Staubli VAL3: MoveLine.pgx

program MoveLine(num x_nX, num x_nY, num x_nZ, num x_nRx, num x_nRy, num x_nRz)
begin
  pPointRx1.trsf.x = x_nX
  pPointRx1.trsf.y = x_nY
  pPointRx1.trsf.z = x_nZ
  pPointRx1.trsf.rx = x_nRx
  pPointRx1.trsf.ry = x_nRy
  pPointRx1.trsf.rz = x_nRz
  movel(pPointRx1,tCurrentTool,mCurrentSpeed)
end
